// TIA Portal V16 export
// export: Created 2021-07-12T14:47:19.7885506Z, ExportSetting WithDefaults, DisplayName Totally Integrated Automation Portal, DisplayVersion V16, DisplayName TIA Portal Version Control Interface, DisplayVersion V16, DisplayName TIA Portal Openness, DisplayVersion V16, DisplayName STEP 7 Professional, DisplayVersion V16, DisplayName STEP 7 Safety, DisplayVersion V16, DisplayName WinCC Professional, DisplayVersion V16
TYPE "LSimaHydTO_typeInternal"
TITLE = LSimaHydTO_typeInternal
// Internal axis data
// stored: IsFailsafeCompliant false
   STRUCT
      Control { S7_SetPoint := 'True'} : "LSimaHydTO_typeInternalControl";   // Command structure, use for axis control
      MotionData { S7_SetPoint := 'True'} : "LSimaHydTO_typeInternalMotionData";   // Motion command data
      PositionLimits_SW { S7_SetPoint := 'True'} : "LSimaHydTO_typePositionLimits";   // Software position limit switch
      UnitsCorrection { S7_SetPoint := 'True'} : "LSimaHydTO_typeInternalUnitsCorrection";   // Correction of units
      CommandIDPool { ExternalAccessible := 'False'; ExternalVisible := 'False'; ExternalWritable := 'False'} : UDInt;   // Source for unique command ID's
   END_STRUCT;
END_TYPE
